// TIA Portal V17 export
// export: Created 2023-05-31T11:26:00.2510914Z, ExportSetting WithDefaults, DisplayName Totally Integrated Automation Portal, DisplayVersion V17, DisplayName TIA Portal Openness, DisplayVersion V17, DisplayName TIA Portal Version Control Interface, DisplayVersion V17, DisplayName STEP 7 Professional, DisplayVersion V17, DisplayName STEP 7 Safety, DisplayVersion V17, DisplayName WinCC Advanced, DisplayVersion V17
VAR_GLOBAL   // PLC tag table "IO_list"
   Input_0 AT %I0.0 : Bool;
   Input_1 AT %I0.1 : Bool;
   Input_2 AT %I0.2 : Bool;
   Input_3 AT %I0.3 : Bool;
   Input_4 AT %I0.4 : Bool;
   Input_5 AT %I0.5 : Bool;
   Input_6 AT %I0.6 : Bool;
   Input_7 AT %I0.7 : Bool;
   Input_8 AT %I1.0 : Bool;
   Input_9 AT %I1.1 : Bool;
   Input_10 AT %I1.2 : Bool;
   Input_11 AT %I1.3 : Bool;
   Input_12 AT %I1.4 : Bool;
   Input_13 AT %I1.5 : Bool;
   Output_0 AT %Q0.0 : Bool;
   Output_1 AT %Q0.1 : Bool;
   Output_2 AT %Q0.2 : Bool;
   Output_3 AT %Q0.3 : Bool;
   Output_4 AT %Q0.4 : Bool;
   Output_5 AT %Q0.5 : Bool;
   Output_6 AT %Q0.6 : Bool;
   Output_7 AT %Q0.7 : Bool;
   Output_8 AT %Q1.0 : Bool;
   Output_9 AT %Q1.1 : Bool;
   AInput_0 AT %IW64 : Int;   // Voltage 0..10V
   AInput_1 AT %IW66 : Int;   // Voltage 0..10V
   AOutput_0 AT %QW64 : Int;   // Current 0..20mA
   AOutput_1 AT %QW66 : Int;   // Current 0..20mA
   AOutput_2 AT %QW80 : Int;   // Voltage 0..10V
END_VAR
